VAR_GLOBAL
	
    {attribute 'pytmc' := '
		pv: TV2K0:VFS:1
	'}
	fb_TV2K0_VFS_1 : FB_VFS;
END_VAR

(* stored: Version 1.1.0.1, ProductVersion 3.1.4024.2
   GVL GVL_SXR_VAC_FS_DEVICES: Id {86bcd696-75bd-4bc1-9d68-0e5f06e66bc8} *)
